///{attribute 'qualified_only'}
VAR_GLOBAL CONSTANT
    MAX_NO_OF_SUBMODULES : UDINT := 20;
    MAX_NO_OF_COMPONENTS : UDINT := 32;

    ePMLUNITMODEDEFAULT : E_PMLUnitMode := E_PMLUnitMode.ePMLUnitMode_Production;
    ePMLSTATEDEFAULT    : E_PMLCommand  := E_PMLCommand.ePMLCommand_Abort;

END_VAR

(* stored: Version 1.1.0.1, ProductVersion 3.1.4024.11
   GVL GVL_PML_Base: Id {88840026-5b28-4ec2-81db-7df0c3fd899b} *)
